// TIA Portal V19 export
FUNCTION_BLOCK "SetPrfOnWork"   // FB9, LAD
TITLE = Activate Profile On Work
// stored: Access Published, MemoryReserve 100, SetENOAutomatically false
   VAR_INPUT
      Enable : Bool;
   END_VAR
   VAR_IN_OUT
      HMI : "Prg_HMI";
      GET_ITF : "Prg_GetITF";
      GET_Data : Variant;
      PRG_Data : Variant;
   END_VAR
   VAR
      GetPrf : "GetPrg";
      tonDone { S7_SetPoint := 'True'} : IEC_TIMER;
   END_VAR
BEGIN

REGION Network 1: Get Profile
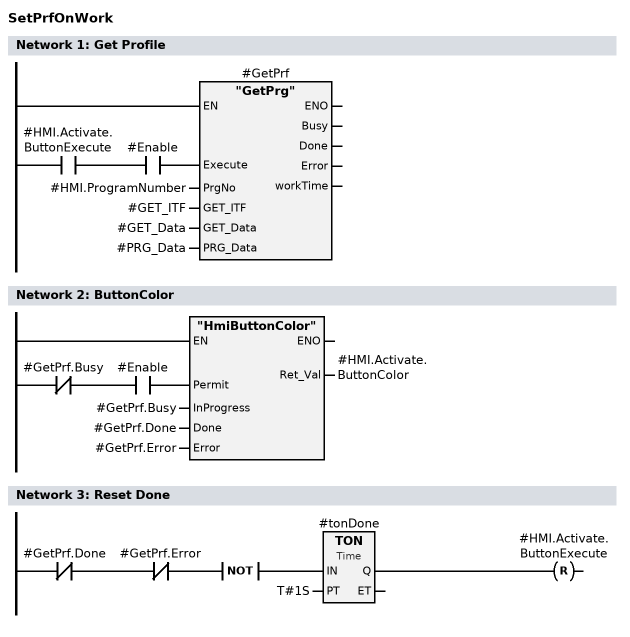
   RUNG wire#powerrail
      #GetPrf(Execute := wire#w1, PrgNo := #HMI.ProgramNumber, GET_ITF := #GET_ITF, GET_Data := #GET_Data, PRG_Data := #PRG_Data, Busy =>, Done =>, Error =>, workTime =>)
   END_RUNG
   RUNG wire#powerrail
      Contact( #HMI.Activate.ButtonExecute )
      Contact( #Enable )
   END_RUNG wire#w1
   // the same network as SCL:
   #GetPrf(Execute := #HMI.Activate.ButtonExecute AND #Enable,   // "GetPrg"
           PrgNo := #HMI.ProgramNumber,
           GET_ITF := #GET_ITF,
           GET_Data := #GET_Data,
           PRG_Data := #PRG_Data);
END_REGION

REGION Network 2: ButtonColor
   RUNG wire#powerrail
      "HmiButtonColor"(Permit := wire#w1, InProgress := #GetPrf.Busy, Done := #GetPrf.Done, Error := #GetPrf.Error, Ret_Val => #HMI.Activate.ButtonColor)
   END_RUNG
   RUNG wire#powerrail
      I_Contact( #GetPrf.Busy )
      Contact( #Enable )
   END_RUNG wire#w1
   // the same network as SCL:
   #HMI.Activate.ButtonColor := "HmiButtonColor"(Permit := NOT #GetPrf.Busy AND #Enable,
                           InProgress := #GetPrf.Busy,
                           Done := #GetPrf.Done,
                           Error := #GetPrf.Error);
END_REGION

REGION Network 3: Reset Done
   RUNG wire#powerrail
      I_Contact( #GetPrf.Done )
      I_Contact( #GetPrf.Error )
      Not()
      { S7_Templates := "time_type := Time" } #tonDone.TON(pt := T#1S, et =>)
      R_Coil( #HMI.Activate.ButtonExecute )
   END_RUNG
   // the same network as SCL:
   #tonDone.TON(IN := NOT (NOT #GetPrf.Done AND NOT #GetPrf.Error), PT := T#1S);
   IF #tonDone.Q THEN #HMI.Activate.ButtonExecute := FALSE; END_IF;
END_REGION
END_FUNCTION_BLOCK
